FUNCTION_BLOCK FB_MCPower EXTENDS MC_Power
VAR_INPUT
    bEnable   : BOOL;      // Enable signal
    bReset    : BOOL;      // Manual reset to clear errors
END_VAR
VAR_OUTPUT
    bActive   : BOOL;      // Indicates if the motor is powered on
    bError    : BOOL;      // Indicates if there is an error
    iErrorID  : UDINT;     // Stores the error ID
	bStatus	  : BOOL;	   // MC_Power Status
END_VAR
VAR_IN_OUT
END_VAR
VAR
    MC_PowerFB  : MC_Power;
    MC_ResetFB  : MC_Reset;
END_VAR

// Check if the axis is already active before enabling
IF bReset THEN
    // Reset errors
    MC_ResetFB(Axis := Axis, Execute := TRUE);
    IF NOT MC_ResetFB.Busy THEN
        bError := FALSE;
        iErrorID := 0;
    END_IF;
ELSIF bEnable THEN
    // Check if already active before enabling
    IF NOT MC_PowerFB.Active THEN
        MC_PowerFB(
            Axis := Axis,
            Enable := TRUE,
            Enable_Positive := TRUE,
            Enable_Negative := TRUE
        );
    END_IF;
END_IF;

// Output states
bActive := MC_PowerFB.Active;
bStatus := MC_PowerFB.Status;
bError := MC_PowerFB.Error;
iErrorID := MC_PowerFB.ErrorID;

END_FUNCTION_BLOCK

(* stored: Version 1.1.0.1, ProductVersion 3.1.4024.12
   POU FB_MCPower: Id {b4d6b702-951d-459e-b23b-a23416a86e07}, SpecialFunc None *)
